// TIA Portal V19 export
DATA_BLOCK "A0303_Manager"   // DB163
// stored: InstanceOfName A0303_Manager_FB, InstanceOfType FB
"A0303_Manager_FB"
   // VAR_INPUT
   //    AreaInterface : "AreaInterface";
   //    DataIn : Struct
   //       LsCheckPassaggio_Coda : Bool;
   //       LsCheckPassaggio_Testa : Bool;
   //       LsPezzoPosMax_Coda : Bool;
   //       LsPezzoPosMax_Testa : Bool;
   //       SemiAut_Pb : Bool;
   //    END_STRUCT;
   //    CIn : Struct
   //       PareggiatoreTesta : Struct
   //          Ax : "Positioning_DOL_Machine_COut";
   //       END_STRUCT;
   //       PareggiatoreCoda : Struct
   //          Ax : "Positioning_DOL_Machine_COut";
   //       END_STRUCT;
   //       Spalle : Struct
   //          Testa : Struct
   //             Ax : "Positioning_DOL_Machine_COut";
   //          END_STRUCT;
   //          Coda : Struct
   //             Ax : "Positioning_DOL_Machine_COut";
   //          END_STRUCT;
   //       END_STRUCT;
   //       Spintore : Struct
   //          Vrt : "ValveMachine_COut";
   //          Orz : "ValveMachine_COut";
   //       END_STRUCT;
   //       TraslazioneStrato : Struct
   //          Ax_Testa : "Positioning_EPOS_Machine_COut";
   //          Ax_Coda : "Positioning_EPOS_Machine_COut";
   //          Manip_Sostegno : "ValveMachine_COut";
   //          Manip_Pareggiatore : "ValveMachine_COut";
   //          SostegnoVrt : "ValveMachine_COut";
   //          IsMeasuring : Bool;
   //       END_STRUCT;
   //       Sollevamento : Struct
   //          Ax_Testa : "Positioning_DOL_Machine_COut";
   //          Ax_Coda : "Positioning_DOL_Machine_COut";
   //       END_STRUCT;
   //       Sostegno : Struct
   //          Testa : Struct
   //             Ax : "Positioning_DOL_Machine_COut";
   //             Paletto : Struct
   //                CtrlSafe : Bool;
   //                Standstill : Bool;
   //                Rest_CheckNext : Bool;
   //                Work_CheckNext : Bool;
   //                Pos : Int;
   //                RestPosition : Bool;
   //             END_STRUCT;
   //          END_STRUCT;
   //          Coda : Struct
   //             Ax : "Positioning_DOL_Machine_COut";
   //             Paletto : Struct
   //                CtrlSafe : Bool;
   //                Standstill : Bool;
   //                Rest_CheckNext : Bool;
   //                Work_CheckNext : Bool;
   //                Pos : Int;
   //                RestPosition : Bool;
   //             END_STRUCT;
   //          END_STRUCT;
   //       END_STRUCT;
   //       Navetta : Struct
   //          ReadyToRecive : Bool;
   //          OutOfWorkspace : Bool;
   //          InPosizioneDiDeposito : Bool;
   //          InPosizioneDiPrelievo : Bool;
   //          InPosizioneDiPrePrelievo : Bool;
   //          RequestDeposito : Bool;
   //          RequestPrelievo : Bool;
   //       END_STRUCT;
   //       ProdManager : "Prod_Beam_Ctrl";
   //    END_STRUCT;
   // END_VAR
   // VAR_OUTPUT
   //    MachineInterface : "MachineInterface";
   //    COut : Struct
   //       Spalla : Struct
   //          Testa : "Positioning_DOL_Machine_Manager";
   //          Coda : "Positioning_DOL_Machine_Manager";
   //       END_STRUCT;
   //       Spintore : Struct
   //          EnableStopDoorOpeningReq : Bool;
   //          EnableStopInPhase : Bool;
   //          EnableStopProgrammed : Bool;
   //          Control_ON : Bool;
   //          CanMoveFreely : Bool;
   //          Rest : Bool;
   //          Work : Bool;
   //       END_STRUCT;
   //       Trasporto : Struct
   //          EnableStopDoorOpeningReq : Bool;
   //          EnableStopInPhase : Bool;
   //          EnableStopProgrammed : Bool;
   //          Control_ON : Bool;
   //          CanMoveFreely : Bool;
   //          OP : Struct
   //             VAI_A_PRELIEVO : Bool;
   //             PRELIEVO : Bool;
   //             VAI_A_DEPOSITO : Bool;
   //             DEPOSITO : Bool;
   //          END_STRUCT;
   //       END_STRUCT;
   //       Sollevatore : Struct
   //          EnableStopDoorOpeningReq : Bool;
   //          EnableStopInPhase : Bool;
   //          EnableStopProgrammed : Bool;
   //          Control_ON : Bool;
   //          CanMoveFreely : Bool;
   //          TargetPosition : LReal;
   //          OP : Struct
   //             PRELIEVO : Bool;
   //             PRE_DEPOSITO : Bool;
   //             DEPOSITO : Bool;
   //          END_STRUCT;
   //       END_STRUCT;
   //       Sostegno : Struct
   //          Testa : Struct
   //             EnableStopDoorOpeningReq : Bool;
   //             EnableStopInPhase : Bool;
   //             EnableStopProgrammed : Bool;
   //             Control_ON : Bool;
   //             CanMoveFreely : Bool;
   //             Phase : Struct
   //                VAI_A_LAVORO : Bool;
   //                VAI_A_RIPOSO : Bool;
   //             END_STRUCT;
   //             Ax : Struct
   //                Pos { ExternalVisible := 'False'; ExternalWritable := 'False'} : LReal;
   //             END_STRUCT;
   //             Paletti : Struct
   //                PosPaletto : Int;
   //                Pos1Collision : Bool;
   //                Pos2Collision : Bool;
   //             END_STRUCT;
   //          END_STRUCT;
   //          Coda : Struct
   //             EnableStopDoorOpeningReq : Bool;
   //             EnableStopInPhase : Bool;
   //             EnableStopProgrammed : Bool;
   //             Control_ON : Bool;
   //             CanMoveFreely : Bool;
   //             Phase : Struct
   //                VAI_A_LAVORO : Bool;
   //                VAI_A_RIPOSO : Bool;
   //             END_STRUCT;
   //             Ax : Struct
   //                Pos { ExternalVisible := 'False'; ExternalWritable := 'False'} : LReal;
   //             END_STRUCT;
   //             Paletti : Struct
   //                PosPaletto : Int;
   //                Pos1Collision : Bool;
   //                Pos2Collision : Bool;
   //             END_STRUCT;
   //          END_STRUCT;
   //       END_STRUCT;
   //       Manipolatore : Struct
   //          ReadyToRecive : Bool;
   //       END_STRUCT;
   //    END_STRUCT;
   // END_VAR
   // VAR_IN_OUT
   //    Par : Struct
   //       Antiribaltamento : Struct
   //          Offset_Pos : LReal;
   //       END_STRUCT;
   //    END_STRUCT;
   //    Par_Trasporto : Struct
   //       PosPrelievo : LReal;
   //       PosDeposito : LReal;
   //       ToleranceWindow : LReal;
   //    END_STRUCT;
   //    Par_Sollevatore : Struct
   //       PosDeposito : LReal;
   //       OffsetPrelievo : LReal;
   //       ToleranceWindow : LReal;
   //    END_STRUCT;
   //    Par_SostegnoAntirib : Struct
   //       RestPosition : LReal;
   //       ToleranceWindow : LReal;
   //       PosTimeout : Time;
   //    END_STRUCT;
   //    Par_Spalla_Testa : Struct
   //       MinDistanzaConParegg : LReal;
   //       ToleranceWindow : LReal;
   //    END_STRUCT;
   //    Par_Spalla_Coda : Struct
   //       MinDistanzaConParegg : LReal;
   //       ToleranceWindow : LReal;
   //    END_STRUCT;
   // END_VAR
   // VAR
   //    Alarm : Struct
   //       TrkPassaggioPezzo : Bool;
   //       TrkPreparationAlreadyFull : Bool;
   //       TrkStackerAlreadyFull : Bool;
   //       PaccoOltreLimiteMax : Bool;
   //       STOP_FineTurno : Bool;
   //       STOP_End_Of_Proroduction : Bool;
   //       STOP_ControlloQualita : Bool;
   //       STOP_Inattività : Bool;
   //    END_STRUCT;
   //    Warning : Struct
   //       IsWaiting_NoPiecesBefore : Bool;
   //       IsWaiting_NoPiecesBefore_A01NotInCycle : Bool;
   //       IsWaiting_NoPiecesBefore_A02NotInCycle : Bool;
   //       IsWaiting_NoPiecesBefore_A03NotInCycle : Bool;
   //       IsWaiting_ShuttleUnload : Bool;
   //       IsWaiting_PezziDaRintegrare : Bool;
   //       STOP_End_Of_Proroduction : Bool;
   //       STOP_FineTurno : Bool;
   //       STOP_ControlloQualita : Bool;
   //       MissingCnd : Struct
   //          SollevatoreNotReadyToRecive : Bool;
   //       END_STRUCT;
   //    END_STRUCT;
   //    OP_CND : Struct
   //       Trasporto : Struct
   //          VaiAPrelievo : Array[0..15] of "OpCnd";
   //          Prelievo { S7_SetPoint := 'True'} : Array[0..15] of "OpCnd";
   //          VaiADeposito : Array[0..15] of "OpCnd";
   //          Deposito : Array[0..15] of "OpCnd";
   //       END_STRUCT;
   //    END_STRUCT;
   //    Ctrl : Struct
   //       Stop : Bool;
   //       Cycle : Struct
   //          Trasferimento : Struct
   //             VaiAPrelievo : Bool;
   //             Prelievo : Bool;
   //             VaiADeposito : Bool;
   //             Deposito : Bool;
   //          END_STRUCT;
   //          Sollevamento : Struct
   //             Prelievo : Bool;
   //             Deposito : Bool;
   //             PreDeposito : Bool;
   //          END_STRUCT;
   //          SostegnoAntirib_Testa : Struct
   //             VaiALavoro : Bool;
   //             VaiARiposo : Bool;
   //             CyclePos : LReal;
   //             PalettoPos : Int;
   //          END_STRUCT;
   //          SostegnoAntirib_Coda : Struct
   //             VaiALavoro : Bool;
   //             VaiARiposo : Bool;
   //             CyclePos : LReal;
   //             PalettoPos : Int;
   //          END_STRUCT;
   //       END_STRUCT;
   //       BTrk : Struct
   //          B3ToLayer1 : Bool;
   //          TransferToStacker : Bool;
   //       END_STRUCT;
   //       Spintore : Struct
   //          Vrt : Struct
   //             Rest : Bool;
   //             Work : Bool;
   //          END_STRUCT;
   //          Orz : Struct
   //             Rest : Bool;
   //             Work : Bool;
   //          END_STRUCT;
   //          Work : Bool;
   //          Rest : Bool;
   //       END_STRUCT;
   //       Spalle : Struct
   //          Testa : Struct
   //             MoveToPos : Bool;
   //             Pos : LReal;
   //          END_STRUCT;
   //          Coda : Struct
   //             MoveToPos : Bool;
   //             Pos : LReal;
   //          END_STRUCT;
   //       END_STRUCT;
   //       TraslazioneStrato : Struct
   //          Ax : Struct
   //             MovePrelievo : Bool;
   //             MoveDeposito : Bool;
   //             PosDeposito : LReal;
   //             PosPrelievo : LReal;
   //          END_STRUCT;
   //          SostegnoVrt : Struct
   //             Rest : Bool;
   //             Work : Bool;
   //          END_STRUCT;
   //          Manip_Sostegno : Struct
   //             Rest : Bool;
   //             Work : Bool;
   //          END_STRUCT;
   //          Manip_Pareggiatore : Struct
   //             Rest : Bool;
   //             Work : Bool;
   //          END_STRUCT;
   //       END_STRUCT;
   //    END_STRUCT;
   //    Sts : Struct
   //       AlarmsPresence : Bool;
   //       WarningsPresence : Bool;
   //       IsStandstill : Bool;
   //       SemiAut : Struct
   //          ON : Bool;
   //          PbMaterialFwd : Bool;
   //          Request : Bool;
   //       END_STRUCT;
   //       SpallaTesta : Struct
   //          InCyclePos : Bool;
   //       END_STRUCT;
   //       SpallaCoda : Struct
   //          InCyclePos : Bool;
   //       END_STRUCT;
   //       Sollevatore : Struct
   //          ReadyToRecive : Bool;
   //          InPrelievoPos : Bool;
   //          InPrePrelievoPos : Bool;
   //          InPosDeposito : Bool;
   //          InPosPreDeposito : Bool;
   //       END_STRUCT;
   //       Preparazione : Struct
   //          Completato : Bool;
   //       END_STRUCT;
   //       TraslazioneStrato : Struct
   //          InPosDeposito : Bool;
   //          InPosPrelievo : Bool;
   //          OutOfWorkspace : Bool;
   //          DropRequest : Bool;
   //       END_STRUCT;
   //       SostegnoTesta : Struct
   //          Ax : Struct
   //             InCyclePos : Bool;
   //             InRestPos : Bool;
   //          END_STRUCT;
   //          Paletto : Struct
   //             InCyclePos : Bool;
   //          END_STRUCT;
   //       END_STRUCT;
   //       SostegnoCoda : Struct
   //          Ax : Struct
   //             InCyclePos : Bool;
   //             InRestPos : Bool;
   //          END_STRUCT;
   //          Paletto : Struct
   //             InCyclePos : Bool;
   //          END_STRUCT;
   //       END_STRUCT;
   //       BTrk { ExternalAccessible := 'False'; ExternalVisible := 'False'; ExternalWritable := 'False'} : Struct
   //          ZonePreparationEmpty { S7_SetPoint := 'True'} : Bool;
   //          ZoneStackerEmpty : Bool;
   //          Actual_O_ID : DInt;
   //       END_STRUCT;
   //    END_STRUCT;
   //    AUX : Struct
   //       LsPosition1Coda_PE { ExternalAccessible := 'False'; ExternalVisible := 'False'; ExternalWritable := 'False'} : Bool;
   //       LsPosition1Coda_NE { ExternalAccessible := 'False'; ExternalVisible := 'False'; ExternalWritable := 'False'} : Bool;
   //       LsPosition1Testa_PE { ExternalAccessible := 'False'; ExternalVisible := 'False'; ExternalWritable := 'False'} : Bool;
   //       LsPosition1Testa_NE { ExternalAccessible := 'False'; ExternalVisible := 'False'; ExternalWritable := 'False'} : Bool;
   //       TrkToTransfer { ExternalAccessible := 'False'; ExternalVisible := 'False'; ExternalWritable := 'False'} : Bool;
   //       TrkToShuttle : Bool;
   //       SemiAut_Pb : Bool;
   //    END_STRUCT;
   //    TON_PassaggioPezzoAlarm : IEC_TIMER;
   //    TON_NoPiecesBefore : IEC_TIMER;
   //    TON_Stop { S7_SetPoint := 'True'} : IEC_TIMER;
   //    TON_StopPerInattivita { S7_SetPoint := 'True'} : IEC_TIMER;
   //    Attrezzamento : Struct
   //       Ready : Bool;
   //       FindNewID : Bool;
   //       RequestNewPosition : Bool;
   //       TargetSpalle : LReal;
   //       TargetSostegno : LReal;
   //       ID : DInt;
   //    END_STRUCT;
   //    CycleWithShortPiece : Bool;
   //    PE_Engaged_Coda : Bool;
   //    NE_Engaged_Coda : Bool;
   //    PE_Engaged_Testa : Bool;
   //    NE_Engaged_Testa : Bool;
   //    TON_CheckCompletato_Stacker : IEC_TIMER;
   //    TON_CheckCompletato_Preparation : IEC_TIMER;
   // END_VAR
BEGIN
END_DATA_BLOCK
